# EPICS substitutions: lsredis/iocBoot/iocLinux/motorSim.substitutions
file "$(MOTOR)/db/asyn_motor.db"
{
pattern
{P,     N,  M,      DTYP,            PORT, ADDR,  DESC,          EGU,      DIR,  VELO,  VBAS,  ACCL,  BDST,  BVEL,  BACC,  MRES,  PREC,  DHLM,  DLLM,  INIT}
{lsredis:,  1,  "m$(N)",  "asynMotor",  motorSim1,  0,  "motor $(N)",  degrees,  Pos,  1,     .1,    .2,    0,     1,     .2,    0.01,  5,     100,   -100,  ""}
{lsredis:,  2,  "m$(N)",  "asynMotor",  motorSim1,  1,  "motor $(N)",  degrees,  Pos,  1,     .1,    .2,    0,     1,     .2,    0.01,  5,     100,   -100,  ""}
{lsredis:,  3,  "m$(N)",  "asynMotor",  motorSim1,  2,  "motor $(N)",  degrees,  Pos,  1,     .1,    .2,    0,     1,     .2,    0.01,  5,     100,   -100,  ""}
{lsredis:,  4,  "m$(N)",  "asynMotor",  motorSim1,  3,  "motor $(N)",  degrees,  Pos,  1,     .1,    .2,    0,     1,     .2,    0.01,  5,     100,   -100,  ""}
{lsredis:,  5,  "m$(N)",  "asynMotor",  motorSim1,  4,  "motor $(N)",  degrees,  Pos,  1,     .1,    .2,    0,     1,     .2,    0.01,  5,     100,   -100,  ""}
{lsredis:,  6,  "m$(N)",  "asynMotor",  motorSim1,  5,  "motor $(N)",  degrees,  Pos,  1,     .1,    .2,    0,     1,     .2,    0.01,  5,     100,   -100,  ""}
{lsredis:,  7,  "m$(N)",  "asynMotor",  motorSim1,  6,  "motor $(N)",  degrees,  Pos,  1,     .1,    .2,    0,     1,     .2,    0.01,  5,     100,   -100,  ""}
{lsredis:,  8,  "m$(N)",  "asynMotor",  motorSim1,  7,  "motor $(N)",  degrees,  Pos,  1,     .1,    .2,    0,     1,     .2,    0.01,  5,     100,   -100,  ""}
{lsredis:,  9,  "m$(N)",  "asynMotor",  motorSim1,  8,  "motor $(N)",  degrees,  Pos,  1,     .1,    .2,    0,     1,     .2,    0.01,  5,     100,   -100,  ""}
{lsredis:,  10,  "m$(N)",  "asynMotor",  motorSim1,  9,  "motor $(N)",  degrees,  Pos,  1,     .1,    .2,    0,     1,     .2,    0.01,  5,     100,   -100,  ""}
{lsredis:,  11,  "m$(N)",  "asynMotor",  motorSim1,  10,  "motor $(N)",  degrees,  Pos,  1,     .1,    .2,    0,     1,     .2,    0.01,  5,     100,   -100,  ""}
{lsredis:,  12,  "m$(N)",  "asynMotor",  motorSim1,  11,  "motor $(N)",  degrees,  Pos,  1,     .1,    .2,    0,     1,     .2,    0.01,  5,     100,   -100,  ""}
{lsredis:,  13,  "m$(N)",  "asynMotor",  motorSim1,  12,  "motor $(N)",  degrees,  Pos,  1,     .1,    .2,    0,     1,     .2,    0.01,  5,     100,   -100,  ""}
{lsredis:,  14,  "m$(N)",  "asynMotor",  motorSim1,  13,  "motor $(N)",  degrees,  Pos,  1,     .1,    .2,    0,     1,     .2,    0.01,  5,     100,   -100,  ""}
{lsredis:,  15,  "m$(N)",  "asynMotor",  motorSim1,  14,  "motor $(N)",  degrees,  Pos,  1,     .1,    .2,    0,     1,     .2,    0.01,  5,     100,   -100,  ""}
{lsredis:,  16,  "m$(N)",  "asynMotor",  motorSim1,  15,  "motor $(N)",  degrees,  Pos,  1,     .1,    .2,    0,     1,     .2,    0.01,  5,     100,   -100,  ""}
}
